FUNCTION_BLOCK CROSSCOMM_PEER_67813986011379A3 (* Service Interface Function Block Type *)
  (* Standard: 61499-2 *)
  (* Version 0.0, 9/22/2017, bababen, nxtControl GmbH, template *)
  PACKAGE Main;
  (* Compiler Cpp nxtControl builtin 1.0 *)
  {SET_ATTRIBUTE(Runtime.FBType.ImplementingType, Runtime.System#DYNGEN_CROSSCOMM_PEER)}
  {SET_ATTRIBUTE(Configuration.GenericFBType.InterfaceParams, Runtime.System#<InterfaceList> <EventOutputs> <Event Name="CNF"> <With Var="LiftRetractedCNF" /> <With Var="LiftExtendedCNF" /> </Event> </EventOutputs> <OutputVars> <VarDeclaration Name="LiftRetractedCNF" Type="BOOL" /> <VarDeclaration Name="LiftExtendedCNF" Type="BOOL" /> </OutputVars> </InterfaceList>)}
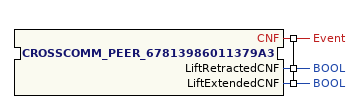
  EVENT_OUTPUT
    CNF WITH LiftRetractedCNF, LiftExtendedCNF;
  END_EVENT
  VAR_OUTPUT
    LiftRetractedCNF : BOOL;
    LiftExtendedCNF : BOOL;
  END_VAR
  EC_STATES
    START;
  END_STATES
END_FUNCTION_BLOCK
